Omron CX-Programmer project NewProject (CX-Programmer 9.75)

# PLC NewPLC1: CP2E-N N

## Global symbols (name address type ; comment)
Actuator_Mie D51 CHANNEL
0 CHANNEL  ; Pick Mie Kering 1
0.00 BOOL  ; Proxy Mie Kering 1
0.01 BOOL  ; PROXY BOWL DISPENSER
0.02 BOOL  ; START BUTTON
0.03 BOOL  ; Proxy Mie Kering 2
0.04 BOOL  ; Proxy Mie Kering 3
0.05 BOOL  ; Proxy Mie Kering 4
0.06 BOOL  ; Proxy Mie Kering 5
0.07 BOOL  ; Proxy Bowl Disp 1
0.08 BOOL  ; Proxy Bowl Disp 2
0.09 BOOL  ; Proxy Bowl Disp 3
1 CHANNEL  ; Pick Bowl 1
100.00 BOOL  ; MOTOR BOWL DISPENSER
100.01 BOOL  ; MOTOR KONVEYOR 1
100.02 BOOL  ; MOTOR KONVEYOR
100.06 BOOL  ; MOTOR LINEAR ACTUATOR 1
100.07 BOOL  ; MOTOR LINEAR ACTUATOR 2
101.00 BOOL  ; MOTOR LINEAR ACTUATOR 3
101.01 BOOL  ; MOTOR LINEAR ACTUATOR 4
101.02 BOOL  ; MOTOR LINEAR ACTUATOR 5
101.03 BOOL  ; Cup Disp 1
101.04 BOOL  ; Cup Disp 2
101.05 BOOL  ; Cup Disp 3
10.02 BOOL  ; Cup Dispensed
200.00 BOOL  ; RELAY START
200.01 BOOL  ; RELAY START KONVEYOR
200.02 BOOL  ; RELAY ACTUATOR
200.03 BOOL  ; MOTOR BOWL
200.04 BOOL  ; RESET COUNTER
C000 BOOL  ; Mie Kering Count
C001 BOOL  ; Cup Count
C003 BOOL  ; StockValidationMie
C004 BOOL  ; Cup_Disp_Cnt
C005 BOOL  ; StockValidationCup
D10 CHANNEL  ; OrderCount
D120 CHANNEL  ; Order Count (From PC)
D5 CHANNEL  ; OrderQty
D6 CHANNEL  ; Order1_Menu
D7 CHANNEL  ; Order2_Menu
D8 CHANNEL  ; Order3_Menu
T000 BOOL  ; TIMER ActuatorMie
T001 BOOL  ; Cycle1 finish
T002 BOOL  ; Reset Second Cup
T003 BOOL  ; Rst Third Cup State
T004 BOOL  ; On MODBUS
T005 BOOL  ; Interlock Linear Actuator retracted
T006 BOOL  ; Timer Boil Mie 1
T007 BOOL  ; Timer Pick Mie Kering 2
T008 BOOL  ; Timer Pick Mie Kering 3
T009 BOOL  ; Timer Boil Mie 2
T010 BOOL  ; Timer Boil Mie 3
W100.02 BOOL  ; Cup_Ready
W100.03 BOOL  ; Boiling_Mie1
W100.04 BOOL  ; Boiling_Mie2
W100.05 BOOL  ; Boiling_Mie3
W100.06 BOOL  ; RebusMie1_Done
W100.07 BOOL  ; RebusMie2_Done
W100.08 BOOL  ; RebusMie3_Done
W100.09 BOOL  ; Start_PickMie2_ToRobot
W100.10 BOOL  ; Start_PickMie3_ToRobot
W100.11 BOOL  ; Order1Topping
W100.12 BOOL  ; Order2Topping
W100.13 BOOL  ; Order3Topping
W101.00 BOOL  ; MieKering1_Ready
W101.01 BOOL  ; MieKering2_Ready
W101.02 BOOL  ; MieKering3_Ready
W101.03 BOOL  ; MieKering4_Ready
W101.04 BOOL  ; MieKering5_Ready
W102.00 BOOL  ; MieKering1 Picked
W102.01 BOOL  ; MieKering2 Picked
W102.02 BOOL  ; MieKering3 Picked
W102.03 BOOL  ; MieKering4 Picked
W102.04 BOOL  ; MieKering5 Picked
W102.05 BOOL  ; Cup1 Ready
W102.06 BOOL  ; Cup2 Ready
W102.07 BOOL  ; Cup3 Ready
W102.08 BOOL  ; Cup1 Picked
W102.09 BOOL  ; Cup2 Picked
W102.10 BOOL  ; Cup3 Picked
W10.00 BOOL  ; RST
W10.01 BOOL  ; MieKering_Picked
W10.02 BOOL  ; Cup dispensed
W10.03 BOOL  ; CupReady
W11.00 BOOL  ; Delay 1sec Trigger
W120.00 BOOL  ; Finished Order From Robot
W125.00 BOOL  ; Reset Stock Mie
W125.01 BOOL  ; Info Kiosk Stock Mie Kosong
W125.02 BOOL  ; Reset Stock Cup
W12.00 BOOL  ; 1 Sec Delay
W1.00 BOOL  ; MieKering_Arrived
W1.01 BOOL  ; MieKering_Picked
W1.02 BOOL  ; Cup_Dropped
W2 CHANNEL  ; Multiple Order States
W20.00 BOOL  ; CheckOrder
W20.05 BOOL  ; Dispensing Done
W22.00 BOOL  ; ON ACTUATOR MIE
W22.01 BOOL  ; ON Actuator Cup
W2.00 BOOL  ; ModbusStatus
W2.01 BOOL  ; TIMRST
W2.02 BOOL  ; 1stOrder Done
W2.03 BOOL  ; Second Cup Done
W2.04 BOOL  ; All Cup Done
W2.05 BOOL  ; ThirdCup
W2.06 BOOL  ; Second Cup
W2.07 BOOL  ; Third Cup Done
W2.08 BOOL  ; LockActuatorMie
W3 CHANNEL  ; Object Position States
W3.00 BOOL  ; StartRelay
W3.01 BOOL  ; MotorMie
W3.02 BOOL  ; Conveyor
W3.03 BOOL  ; Mie Sampe
W3.05 BOOL  ; BowlJatuh
W3.06 BOOL  ; Bowl Arrived
W3.07 BOOL  ; Second Cup
W4.00 BOOL  ; CupDisp Working
W5.00 BOOL  ; Start MODBUS
Cup1_Picked W21.03 BOOL
Cup2_Picked W21.04 BOOL
Cup3_Picked W21.05 BOOL
DispenserMieCnt C002 BOOL
FB_MODBUSTCP_SERVER _CP2E003_ExecuteModTcpServer
MieKering1_Picked W21.00 BOOL
MieKering2_Picked W21.01 BOOL
MieKering3_Picked W21.02 BOOL
Order1_Menu D110 CHANNEL
Order1_Topping1 D100 CHANNEL
Order1_Topping2 D101 CHANNEL
Order1_Topping3 D102 CHANNEL
Order2_Menu D111 CHANNEL
Order2_Topping1 D103 CHANNEL
Order2_Topping2 D104 CHANNEL
Order2_Topping3 D105 CHANNEL
Order3_Menu D112 CHANNEL
Order3_Topping1 D106 CHANNEL
Order3_Topping2 D107 CHANNEL
Order3_Topping3 D108 CHANNEL
Start_Order W100.00 BOOL
StepNum D50 CHANNEL  ; Step Number
Timer_10Sec T011 BOOL  ; 10Sec Delay

## Program CookingMie (cyclic task 0)
Local symbols
p_LT BOOL
p_eq BOOL
p_gt BOOL
p_lt BOOL

### Section MODBUS

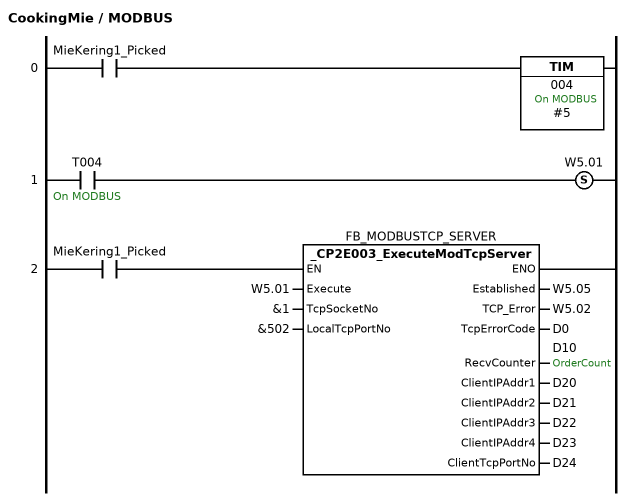
; rung 0
LD MieKering1_Picked
TIM 004 #5  ; On MODBUS
; rung 1
LD T004  ; On MODBUS
SET W5.01
; rung 2
LD MieKering1_Picked
CALL FB_MODBUSTCP_SERVER : _CP2E003_ExecuteModTcpServer (Execute := W5.01, TcpSocketNo := &1, LocalTcpPortNo := &502, Established => W5.05, TCP_Error => W5.02, TcpErrorCode => D0, RecvCounter => D10, ClientIPAddr1 => D20, ClientIPAddr2 => D21, ClientIPAddr3 => D22, ClientIPAddr4 => D23, ClientTcpPortNo => D24)  ; OrderCount

### Section Feeder_Main

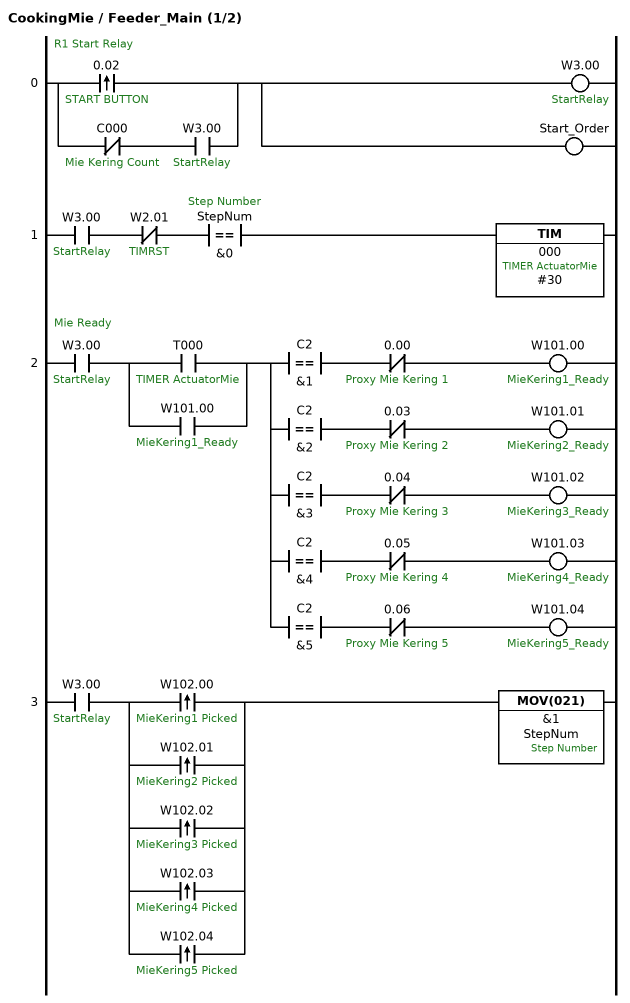
; rung 0: R1 Start Relay
@LD 0.02  ; START BUTTON
LDNOT C000  ; Mie Kering Count
AND W3.00  ; StartRelay
ORLD
OUT W3.00  ; StartRelay
OUT Start_Order
; rung 1
LD W3.00  ; StartRelay
ANDNOT W2.01  ; TIMRST
AND=(300) StepNum &0  ; Step Number
TIM 000 #30  ; TIMER ActuatorMie
; rung 2: Mie Ready
LD W3.00  ; StartRelay
LD T000  ; TIMER ActuatorMie
OR W101.00  ; MieKering1_Ready
ANDLD
OUT TR0
AND=(300) C2 &1
ANDNOT 0.00  ; Proxy Mie Kering 1
OUT W101.00  ; MieKering1_Ready
LD TR0
AND=(300) C2 &2
ANDNOT 0.03  ; Proxy Mie Kering 2
OUT W101.01  ; MieKering2_Ready
LD TR0
AND=(300) C2 &3
ANDNOT 0.04  ; Proxy Mie Kering 3
OUT W101.02  ; MieKering3_Ready
LD TR0
AND=(300) C2 &4
ANDNOT 0.05  ; Proxy Mie Kering 4
OUT W101.03  ; MieKering4_Ready
LD TR0
AND=(300) C2 &5
ANDNOT 0.06  ; Proxy Mie Kering 5
OUT W101.04  ; MieKering5_Ready
; rung 3
LD W3.00  ; StartRelay
@LD W102.00  ; MieKering1 Picked
@OR W102.01  ; MieKering2 Picked
@OR W102.02  ; MieKering3 Picked
@OR W102.03  ; MieKering4 Picked
@OR W102.04  ; MieKering5 Picked
ANDLD
MOV(021) &1 StepNum  ; Step Number

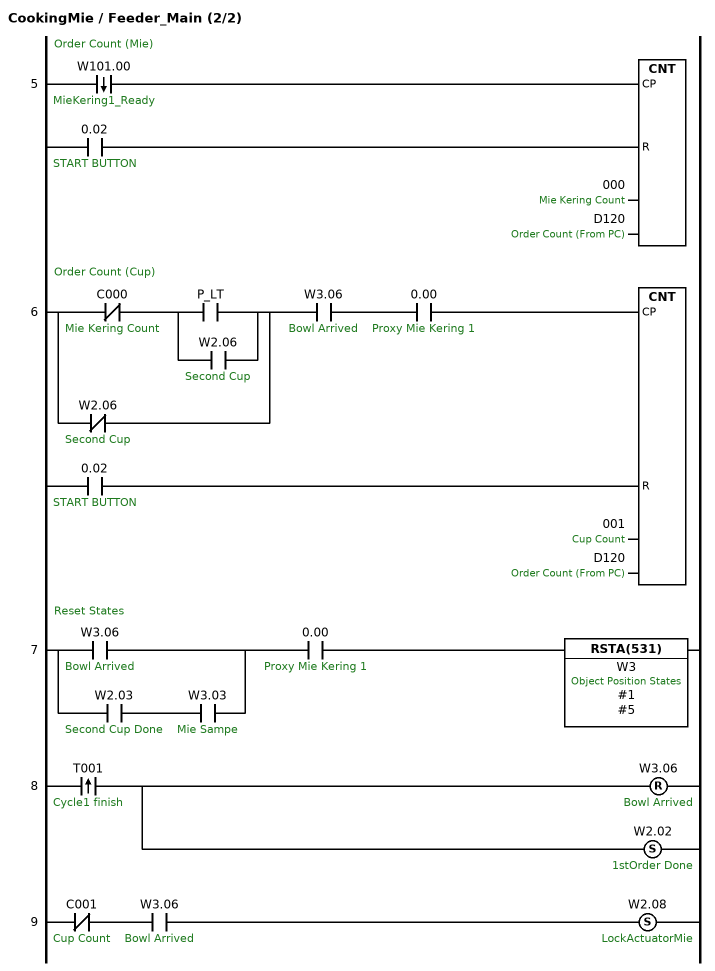
; rung 5: Order Count (Mie)
%LD W101.00  ; MieKering1_Ready
LD 0.02  ; START BUTTON
CNT 000 D120  ; Order Count (From PC), Mie Kering Count
; rung 6: Order Count (Cup)
LDNOT C000  ; Mie Kering Count
LD P_LT
OR W2.06  ; Second Cup
ANDLD
ORNOT W2.06  ; Second Cup
AND W3.06  ; Bowl Arrived
AND 0.00  ; Proxy Mie Kering 1
LD 0.02  ; START BUTTON
CNT 001 D120  ; Order Count (From PC), Cup Count
; rung 7: Reset States
LD W3.06  ; Bowl Arrived
LD W2.03  ; Second Cup Done
AND W3.03  ; Mie Sampe
ORLD
AND 0.00  ; Proxy Mie Kering 1
RSTA(531) W3 #1 #5  ; Object Position States
; rung 8
@LD T001  ; Cycle1 finish
RSET W3.06  ; Bowl Arrived
SET W2.02  ; 1stOrder Done
; rung 9
LDNOT C001  ; Cup Count
AND W3.06  ; Bowl Arrived
SET W2.08  ; LockActuatorMie

### Section Dispenser_Mie

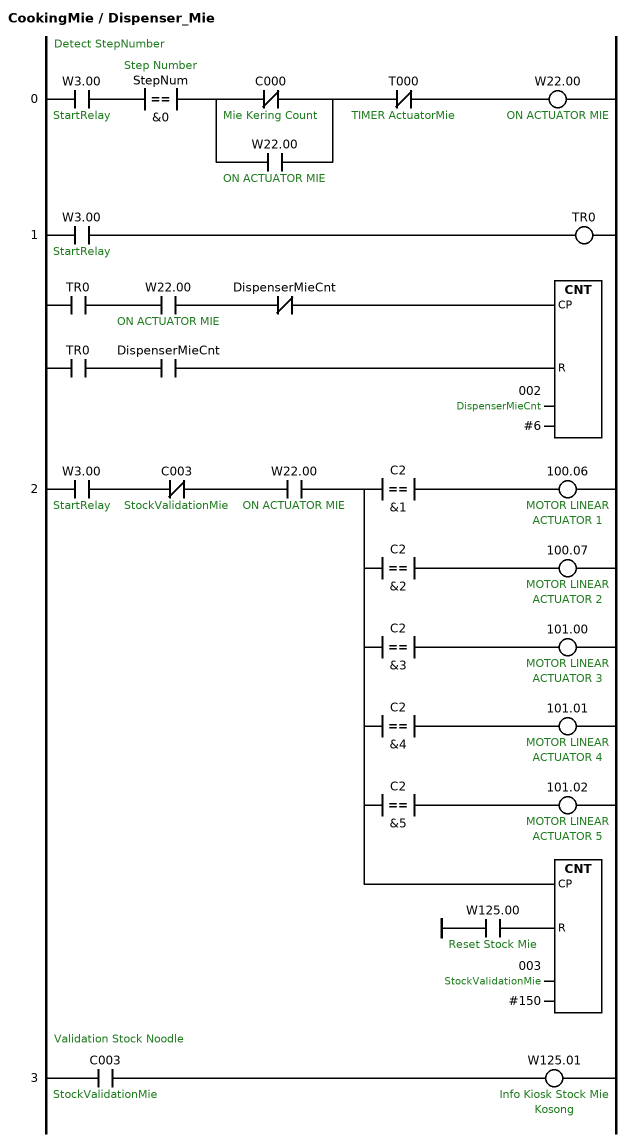
; rung 0: Detect StepNumber
LD W3.00  ; StartRelay
AND=(300) StepNum &0  ; Step Number
LDNOT C000  ; Mie Kering Count
OR W22.00  ; ON ACTUATOR MIE
ANDLD
ANDNOT T000  ; TIMER ActuatorMie
OUT W22.00  ; ON ACTUATOR MIE
; rung 1
LD W3.00  ; StartRelay
OUT TR0
AND W22.00  ; ON ACTUATOR MIE
ANDNOT DispenserMieCnt
LD TR0
AND DispenserMieCnt
CNT 002 #6  ; DispenserMieCnt
; rung 2
LD W3.00  ; StartRelay
ANDNOT C003  ; StockValidationMie
AND W22.00  ; ON ACTUATOR MIE
OUT TR0
AND=(300) C2 &1
OUT 100.06  ; MOTOR LINEAR ACTUATOR 1
LD TR0
AND=(300) C2 &2
OUT 100.07  ; MOTOR LINEAR ACTUATOR 2
LD TR0
AND=(300) C2 &3
OUT 101.00  ; MOTOR LINEAR ACTUATOR 3
LD TR0
AND=(300) C2 &4
OUT 101.01  ; MOTOR LINEAR ACTUATOR 4
LD TR0
AND=(300) C2 &5
OUT 101.02  ; MOTOR LINEAR ACTUATOR 5
LD TR0
LD W125.00  ; Reset Stock Mie
CNT 003 #150  ; StockValidationMie
; rung 3: Validation Stock Noodle
LD C003  ; StockValidationMie
OUT W125.01  ; Info Kiosk Stock Mie Kosong

### Section Dispenser_Cup

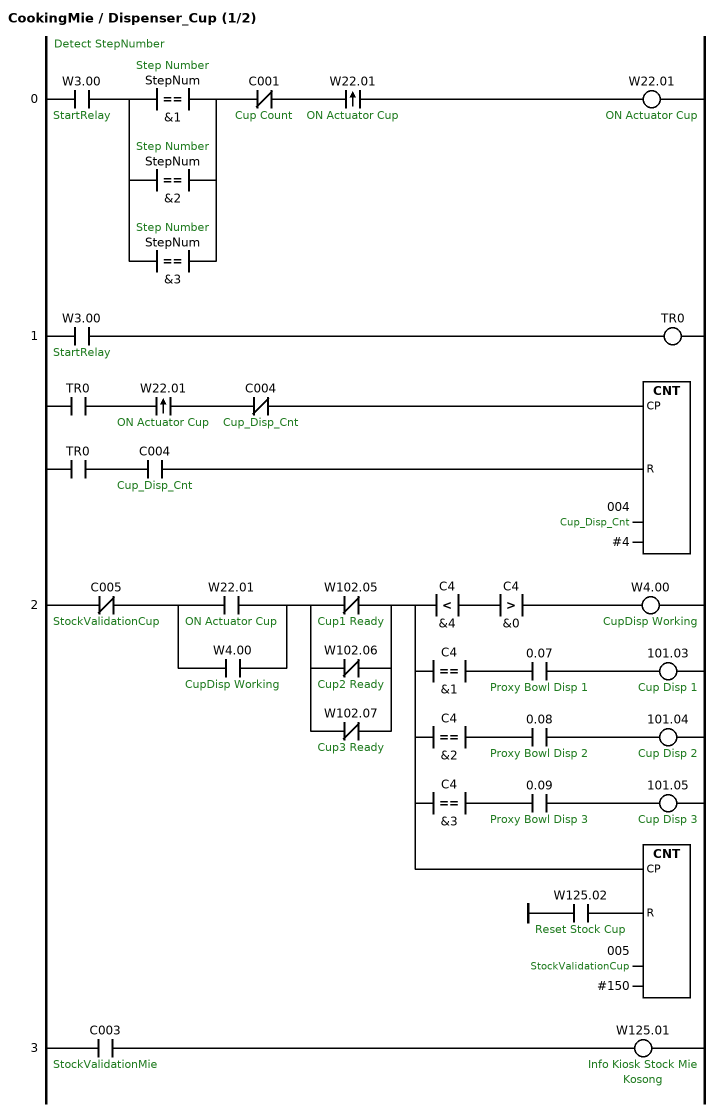
; rung 0: Detect StepNumber
LD W3.00  ; StartRelay
LD=(300) StepNum &1  ; Step Number
OR=(300) StepNum &2  ; Step Number
OR=(300) StepNum &3  ; Step Number
ANDLD
ANDNOT C001  ; Cup Count
@AND W22.01  ; ON Actuator Cup
OUT W22.01  ; ON Actuator Cup
; rung 1
LD W3.00  ; StartRelay
OUT TR0
@AND W22.01  ; ON Actuator Cup
ANDNOT C004  ; Cup_Disp_Cnt
LD TR0
AND C004  ; Cup_Disp_Cnt
CNT 004 #4  ; Cup_Disp_Cnt
; rung 2
LDNOT C005  ; StockValidationCup
LD W22.01  ; ON Actuator Cup
OR W4.00  ; CupDisp Working
ANDLD
LDNOT W102.05  ; Cup1 Ready
ORNOT W102.06  ; Cup2 Ready
ORNOT W102.07  ; Cup3 Ready
ANDLD
OUT TR0
AND<(310) C4 &4
AND>(320) C4 &0
OUT W4.00  ; CupDisp Working
LD TR0
AND=(300) C4 &1
AND 0.07  ; Proxy Bowl Disp 1
OUT 101.03  ; Cup Disp 1
LD TR0
AND=(300) C4 &2
AND 0.08  ; Proxy Bowl Disp 2
OUT 101.04  ; Cup Disp 2
LD TR0
AND=(300) C4 &3
AND 0.09  ; Proxy Bowl Disp 3
OUT 101.05  ; Cup Disp 3
LD TR0
LD W125.02  ; Reset Stock Cup
CNT 005 #150  ; StockValidationCup
; rung 3
LD C003  ; StockValidationMie
OUT W125.01  ; Info Kiosk Stock Mie Kosong

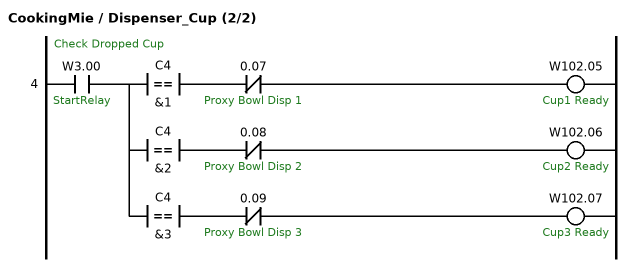
; rung 4: Check Dropped Cup
LD W3.00  ; StartRelay
OUT TR0
AND=(300) C4 &1
ANDNOT 0.07  ; Proxy Bowl Disp 1
OUT W102.05  ; Cup1 Ready
LD TR0
AND=(300) C4 &2
ANDNOT 0.08  ; Proxy Bowl Disp 2
OUT W102.06  ; Cup2 Ready
LD TR0
AND=(300) C4 &3
ANDNOT 0.09  ; Proxy Bowl Disp 3
OUT W102.07  ; Cup3 Ready

### Section Feeder_MultiOrder

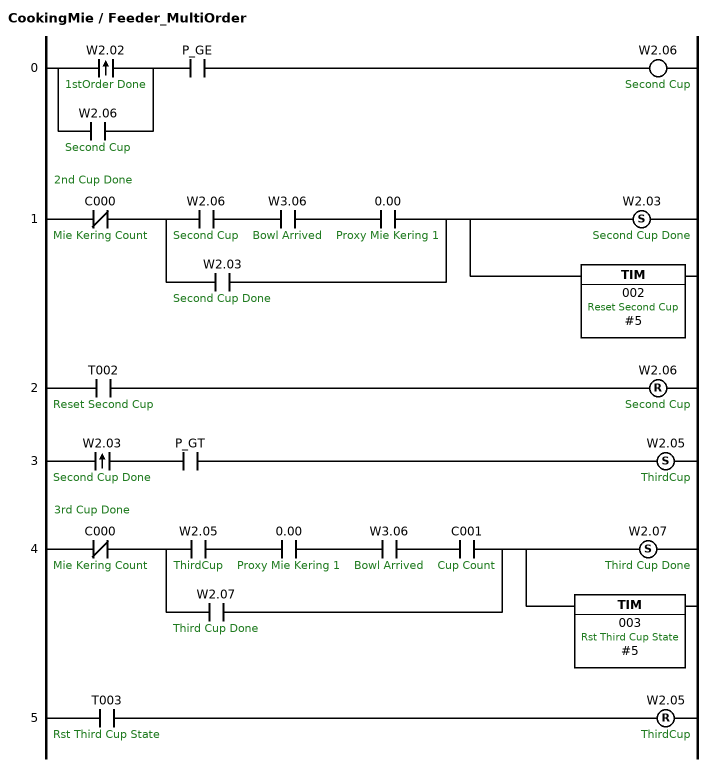
; rung 0
@LD W2.02  ; 1stOrder Done
OR W2.06  ; Second Cup
AND P_GE
OUT W2.06  ; Second Cup
; rung 1: 2nd Cup Done
LDNOT C000  ; Mie Kering Count
LD W2.06  ; Second Cup
AND W3.06  ; Bowl Arrived
AND 0.00  ; Proxy Mie Kering 1
OR W2.03  ; Second Cup Done
ANDLD
SET W2.03  ; Second Cup Done
TIM 002 #5  ; Reset Second Cup
; rung 2
LD T002  ; Reset Second Cup
RSET W2.06  ; Second Cup
; rung 3
@LD W2.03  ; Second Cup Done
AND P_GT
SET W2.05  ; ThirdCup
; rung 4: 3rd Cup Done
LDNOT C000  ; Mie Kering Count
LD W2.05  ; ThirdCup
AND 0.00  ; Proxy Mie Kering 1
AND W3.06  ; Bowl Arrived
AND C001  ; Cup Count
OR W2.07  ; Third Cup Done
ANDLD
SET W2.07  ; Third Cup Done
TIM 003 #5  ; Rst Third Cup State
; rung 5
LD T003  ; Rst Third Cup State
RSET W2.05  ; ThirdCup

### Section Cooking_Process

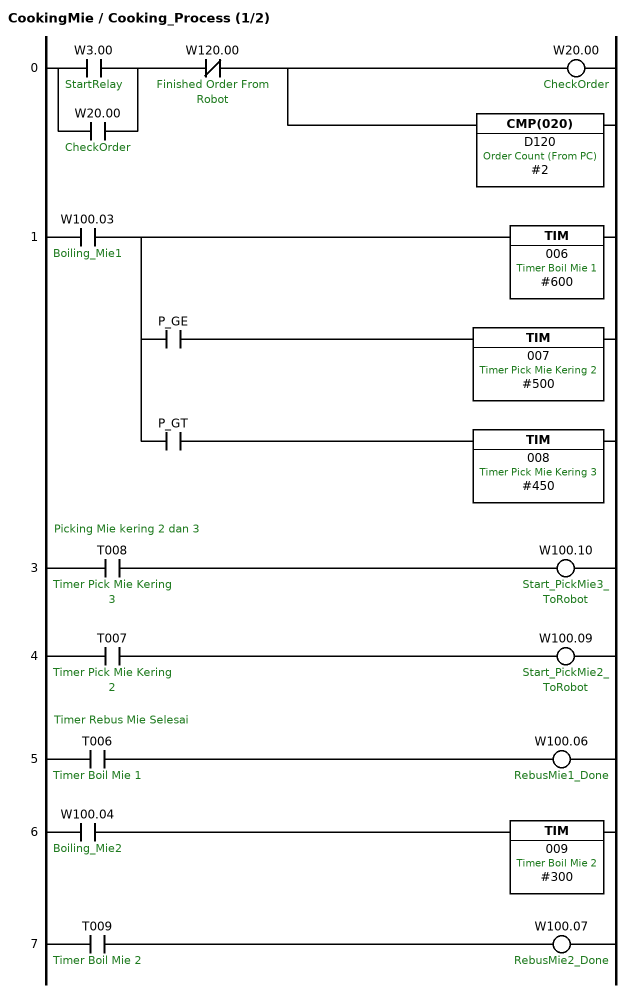
; rung 0
LD W3.00  ; StartRelay
OR W20.00  ; CheckOrder
ANDNOT W120.00  ; Finished Order From Robot
OUT W20.00  ; CheckOrder
CMP(020) D120 #2  ; Order Count (From PC)
; rung 1
LD W100.03  ; Boiling_Mie1
OUT TR0
TIM 006 #600  ; Timer Boil Mie 1
AND P_GE
TIM 007 #500  ; Timer Pick Mie Kering 2
LD TR0
AND P_GT
TIM 008 #450  ; Timer Pick Mie Kering 3
; rung 3: Picking Mie kering 2 dan 3
LD T008  ; Timer Pick Mie Kering 3
OUT W100.10  ; Start_PickMie3_ToRobot
; rung 4
LD T007  ; Timer Pick Mie Kering 2
OUT W100.09  ; Start_PickMie2_ToRobot
; rung 5: Timer Rebus Mie Selesai
LD T006  ; Timer Boil Mie 1
OUT W100.06  ; RebusMie1_Done
; rung 6
LD W100.04  ; Boiling_Mie2
TIM 009 #300  ; Timer Boil Mie 2
; rung 7
LD T009  ; Timer Boil Mie 2
OUT W100.07  ; RebusMie2_Done

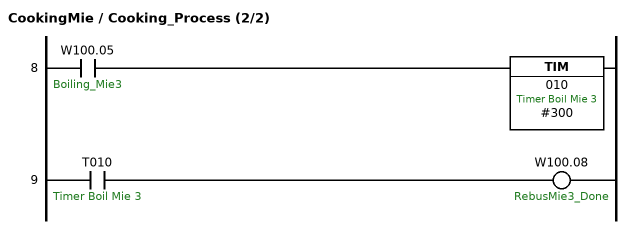
; rung 8
LD W100.05  ; Boiling_Mie3
TIM 010 #300  ; Timer Boil Mie 3
; rung 9
LD T010  ; Timer Boil Mie 3
OUT W100.08  ; RebusMie3_Done

### Section Order_Settings

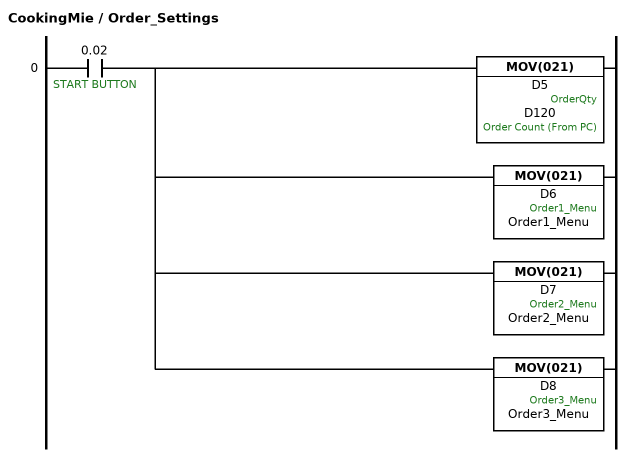
; rung 0
LD 0.02  ; START BUTTON
MOV(021) D5 D120  ; OrderQty, Order Count (From PC)
MOV(021) D6 Order1_Menu  ; Order1_Menu
MOV(021) D7 Order2_Menu  ; Order2_Menu
MOV(021) D8 Order3_Menu  ; Order3_Menu

### Section RESET_States

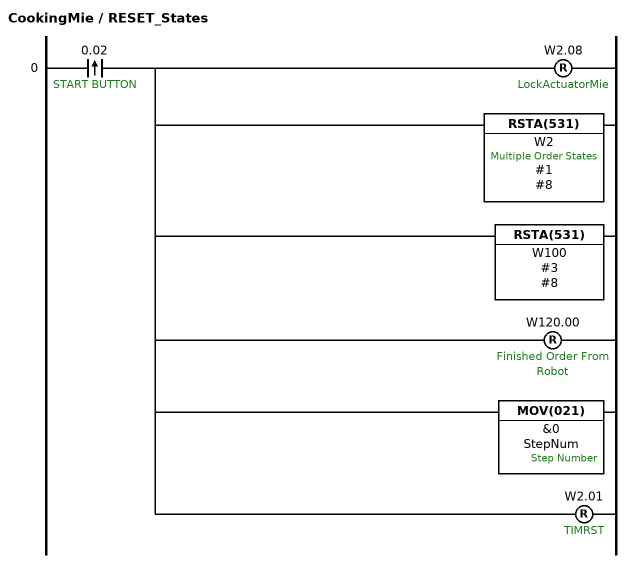
; rung 0
@LD 0.02  ; START BUTTON
RSET W2.08  ; LockActuatorMie
RSTA(531) W2 #1 #8  ; Multiple Order States
RSTA(531) W100 #3 #8
RSET W120.00  ; Finished Order From Robot
MOV(021) &0 StepNum  ; Step Number
RSET W2.01  ; TIMRST

### Section END
; rung 0
END(001)

## Function block _CP2E003_ExecuteModTcpServer (Omron library block, body left out)